PROGRAM MAIN
VAR
END_VAR

END_PROGRAM

(* stored: Version 1.1.0.1
   POU MAIN: Id {ed56dcfa-6359-46ce-be08-022fc3b39b08}, SpecialFunc None *)
